# EPICS substitutions: iocBoot/ioc4idVCDM/substitutions/canberra_13.substitutions
file "$(MCA)/mcaApp/Db/simple_mca.db"
{
pattern
{P           M       DTYP           INP         PREC  CHANS}
{4idVCDM:med:   mca1  "asynMCA"   "@asyn(AIM2/1 0)"    3  2048}
{4idVCDM:med:   mca2  "asynMCA"   "@asyn(AIM2/1 1)"    3  2048}
{4idVCDM:med:   mca3  "asynMCA"   "@asyn(AIM2/1 2)"    3  2048}
{4idVCDM:med:   mca4  "asynMCA"   "@asyn(AIM2/2 0)"    3  2048}
{4idVCDM:med:   mca5  "asynMCA"   "@asyn(AIM2/2 1)"    3  2048}
{4idVCDM:med:   mca6  "asynMCA"   "@asyn(AIM2/2 2)"    3  2048}
{4idVCDM:med:   mca7  "asynMCA"   "@asyn(AIM3/1 0)"    3  2048}
{4idVCDM:med:   mca8  "asynMCA"   "@asyn(AIM3/1 1)"    3  2048}
{4idVCDM:med:   mca9  "asynMCA"   "@asyn(AIM3/1 2)"    3  2048}
{4idVCDM:med:   mca10 "asynMCA"   "@asyn(AIM3/2 0)"    3  2048}
{4idVCDM:med:   mca11 "asynMCA"   "@asyn(AIM3/3 1)"    3  2048}
{4idVCDM:med:   mca12 "asynMCA"   "@asyn(AIM3/4 2)"    3  2048}
{4idVCDM:med:   mca13 "asynMCA"   "@asyn(AIM3/2 3)"    3  2048}
{4idVCDM:med:   mca0  "Soft Channel"   ""     3  2048}
}

file "$(MCA)/mcaApp/Db/icb_amp.db"
{
pattern
{P			AMP		PORT}
{4idVCDM:med:	amp1	"icbAmp1"}
{4idVCDM:med:	amp2	"icbAmp2"}
{4idVCDM:med:	amp3	"icbAmp3"}
{4idVCDM:med:	amp4	"icbAmp4"}
{4idVCDM:med:	amp5	"icbAmp5"}
{4idVCDM:med:	amp6	"icbAmp6"}
{4idVCDM:med:	amp7	"icbAmp7"}
{4idVCDM:med:	amp8	"icbAmp8"}
{4idVCDM:med:	amp9	"icbAmp9"}
{4idVCDM:med:	amp10	"icbAmp10"}
{4idVCDM:med:	amp11	"icbAmp11"}
{4idVCDM:med:	amp12	"icbAmp12"}
{4idVCDM:med:	amp13	"icbAmp13"}
}

file "$(MCA)/mcaApp/Db/icb_adc.db"
{
pattern
{P			ADC		PORT}
{4idVCDM:med:	adc1	"icbAdc1"}
{4idVCDM:med:	adc2	"icbAdc2"}
{4idVCDM:med:	adc3	"icbAdc3"}
{4idVCDM:med:	adc4	"icbAdc4"}
}

file "$(MCA)/mcaApp/Db/icb_hvps.db"
{
pattern
{P			HVPS	LIMIT	PORT}
{4idVCDM:med:	hvps1	1000	"icbHvps1"}
}
